{attribute 'qualified_only'}
{attribute 'strict'}
{attribute 'conditionalshow'}
TYPE eByteOrder :
(
	{attribute 'hide'}
	eBigEndian	:= 0,
	{attribute 'hide'}
	eLittleEndian	:= 1
);
END_TYPE

(* stored: Version 1.1.0.1, ProductVersion 3.1.4024.9
   DUT eByteOrder: Id {a2224297-1b72-4e52-b7cc-00a73ec0090d} *)
